{attribute 'linkalways'} 
{attribute 'no_explicit_call' := 'This FB is a CLASS and must be accessed using methods or properties'}
{attribute 'enable_dynamic_creation'}
FUNCTION_BLOCK Node_F_VN_GetAt_TcVnPoint2_LREAL EXTENDS VisionNode
VAR
    ipContainer : _ITcVnContainer;
    aElement : _TcVnPoint2_LREAL;
    nIndex : _ULINT(0);
    hrPrev : _HRESULT(S_OK);
    hresult : _HRESULT(S_OK);
END_VAR

METHOD PUBLIC  Clone : I_Node
VAR
	pNode : POINTER TO Node_F_VN_GetAt_TcVnPoint2_LREAL;
END_VAR
pNode := __NEW(Node_F_VN_GetAt_TcVnPoint2_LREAL);
Clone := pNode^;
END_METHOD

METHOD FB_init : BOOL
VAR_INPUT
	bInitRetains : BOOL; // if TRUE, the retain variables are initialized (warm start / cold start)
	bInCopyCode : BOOL;  // if TRUE, the instance afterwards gets moved into the copy code (online change)
END_VAR
AddInput('ipContainer', ipContainer);
AddParameter('nIndex', nIndex);
AddInput('hrPrev', hrPrev);
AddOutput('aElement', aElement);
AddOutput('hresult',hresult);
END_METHOD

METHOD PROTECTED OnExecute
hresult.Value := F_VN_GetAt_TcVnPoint2_LREAL(
    ipContainer := ipContainer.Value,
    aElement := aElement.Value,
    nIndex := nIndex.Value,
    hrPrev:= hrPrev.Value);
END_METHOD

METHOD PUBLIC PreExecutionCheck
VAR_INPUT
	Check : I_PreExecutionChecks;
END_VAR
Check.IsTrue(ipContainer.IsValid, 'ipContainer must be a valid container');
Check.IsTrue(ipContainer.IsType(TC_GLOBAL_CONST_LIST.ContainerType_Vector_TcVnPoint2_LREAL), 'ipContainer contains incorrect type');
END_METHOD

END_FUNCTION_BLOCK

(* stored: Version 1.1.0.1, ProductVersion 3.1.4026.13
   POU Node_F_VN_GetAt_TcVnPoint2_LREAL: Id {d3b3b703-c531-4636-87fc-1d554561f65a}, SpecialFunc None
   Folder Constructor: Id {8c9e3a8f-6e43-4468-b87b-2b5a6d78bf3e}
   Method Clone: Id {41d531c9-8d21-4aba-b0be-a6260754d555}
   Method FB_init: Id {f8ab2259-761e-458c-9944-950efc15a6ac}
   Method OnExecute: Id {e037aa46-006d-49ed-8b3d-b09a7682cd37}
   Method PreExecutionCheck: Id {a18f22e7-2d9d-46c3-a687-f1a688df7a33} *)
